(*
Standard control for FB_AxisRef
*)

FUNCTION_BLOCK ABSTRACT FB_AxisControl
VAR_INPUT
END_VAR
VAR_OUTPUT
END_VAR
VAR
END_VAR

END_FUNCTION_BLOCK

(* stored: Version 1.1.0.1, ProductVersion 3.1.4024.12
   POU FB_AxisControl: Id {5be60846-58a1-496b-ab38-aa8e689397e9}, SpecialFunc None *)
